// TIA Portal V18 export
FUNCTION "AOvar" : Void   // FC10011, LAD
{ S7_Optimized_Access := 'TRUE' }
VERSION : 0.1
// stored: AutoNumber false, IsIECCheckEnabled false, SetENOAutomatically false, UDAEnableTagReadback false
   VAR_INPUT
      iFuncSystem : Byte;
      iFuncVar : Byte;
   END_VAR
   VAR_OUTPUT
      rOutput : Real;
   END_VAR
BEGIN

REGION Network 1 (SCL)
   CASE #iFuncSystem OF
       0:  // Statement section case 2 to 4
           ;
       1..4:  // Statement section case 1
           CASE #iFuncVar OF
               0:  // 
                   ;
               1:  // 
                   #rOutput := "AHUAO".AO.rSAFAnalog[#iFuncSystem];
               2:  // 
                   #rOutput := "AHUAO".AO.rHeater[#iFuncSystem];
               3:  // 
                   #rOutput := "AHUAO".AO.rMixingAirDumper[#iFuncSystem];
               4:  // 
                   #rOutput := "AHUAO".AO.rExtractAirDumper[#iFuncSystem];
               5:  // 
                   #rOutput := "AHUAO".AO.rCooler[#iFuncSystem];
               6:  // 
                   #rOutput := "AHUAO".AO.rWHU[#iFuncSystem];
           END_CASE;
       5..9:
           ;
       10: // HS+HC    
           CASE #iFuncVar OF
               0:  // 
                   ;
               1:  //         
                   #rOutput := "HCsAO".AO.rHC3vwCtrl[1];
               2:  //         
                   #rOutput := "HCsAO".AO.rHC3vwCtrl[2];
           END_CASE;
       11..20:
           ;
       21: //Proxy Channels    
           CASE #iFuncVar OF
               0:  //
                   ;
               1..8:  //
                   #rOutput := "AHUProxyCH".Vars.rCHProxySignal[#iFuncVar];
               ELSE
                   ;
           END_CASE;
       ELSE  // Statement section ELSE
           ;
   END_CASE;
END_REGION
END_FUNCTION
